// TIA Portal V19 export
TYPE "TExtEncoder_StatusWord"
// stored: Access Published
   STRUCT
      Enable : Bool;
      Error : Bool;
      RestartActive : Bool;
      OnlineStartValuesChanged : Bool;
      HomingDone : Bool;
      Done : Bool;
      HomingCommand : Bool;
   END_STRUCT;
END_TYPE
